(* PLC project Tc2_Utilities.Int64Add64Ex Demo, tc3-libraries-kb TwinCAT 3.1 *)
(* stored: creationDateTime 2026-05-10T17:00:00, modificationDateTime 2026-05-10T17:00:00 *)

PROGRAM P_Demo_Int64Add64Ex
  VAR
    rResult : T_LARGE_INTEGER;  (* Int64Add64Ex 返回值 *)
    bRun : BOOL;  (* 触发一次调用 *)
    a : T_LARGE_INTEGER;  (* 测试用本地变量 *)
    b : T_LARGE_INTEGER;  (* 测试用本地变量 *)
    bOV : BOOL;  (* 测试用本地变量 *)
  END_VAR

            // ============================================================
// Tc2_Utilities.Int64Add64Ex 演示程序（FUNCTION）
// ============================================================
// 验证步骤：
//   1. 引用 Tc2_Utilities
//   2. 编译 + 登录
//   3. 强制 bRun := TRUE 一个周期
//   4. 在线监视 rResult
// ============================================================

a := LARGE_INTEGER(16#7FFFFFFF, 16#FFFFFFFF); b := LARGE_INTEGER(0, 1);
IF bRun THEN
    rResult := Int64Add64Ex(augend := a, addend := b, bOV := bOV);
    bRun := FALSE;
END_IF;

          
END_PROGRAM
